FUNCTION_BLOCK COMMCHANNELUDPRECV (* Service Interface Function Block Type *)
  (* Standard: 61499-2 *)
  (* Version 0.0, 9/14/2008, Horst Mayer, nxtControl GmbH, template *)
  PACKAGE IEC61499;
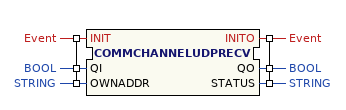
  EVENT_INPUT
    INIT WITH QI, OWNADDR;
  END_EVENT
  EVENT_OUTPUT
    INITO WITH QO, STATUS;
  END_EVENT
  VAR_INPUT
    QI : BOOL;
    OWNADDR : STRING;
  END_VAR
  VAR_OUTPUT
    QO : BOOL; (* Event Output Qualifier *)
    STATUS : STRING;
  END_VAR
END_FUNCTION_BLOCK
